TYPE ProgramaEjecucion :
STRUCT
	EjeX : UINT;
	EjeY : UINT;
	EjeZ : UINT;
	EjeJ : LREAL;
	CoordenadaEjeX : LREAL;
	CoordenadaEjeY : LREAL;
	CoordenadaEjeZ : LREAL;
	CoordenadaEjeJ : LREAL;
END_STRUCT
END_TYPE

(* stored: Version 1.1.0.1, ProductVersion 3.1.4024.11
   DUT ProgramaEjecucion: Id {3b33b89f-26b1-4385-b9e9-5cf7254ffe52} *)
